FUNCTION_BLOCK EL5122
VAR
	_io : EL5122_Data;
	{attribute addProperty Name "WcState"}
	_wcState : WcStateInputToggle;
	{attribute addProperty Name "Info data"}
	_infoData : InfoDataAdsDC;
END_VAR

PROPERTY IO : REFERENCE TO EL5122_Data
GET
IO REF= _io;
END_GET
END_PROPERTY

PROPERTY WcState : REFERENCE TO WcStateInputToggle
GET
WcState REF= _wcState;
END_GET
END_PROPERTY

END_FUNCTION_BLOCK

(* stored: Version 1.1.0.1, ProductVersion 3.1.4024.9
   POU EL5122: Id {14cfafe3-91b0-0d6a-0ec5-621a855ae5fb}, SpecialFunc None
   Property IO: Id {6432d7fb-7653-0cdb-041f-810b7e1d7652}
   Get Get: Id {c6f12ab3-6181-0d9a-17a0-6c7f106cfa6d}
   Property WcState: Id {62db1900-afe2-0547-214a-f9538e2d305e}
   Get Get: Id {8eef0600-efd9-062e-2e22-aa57533eac4b} *)
